FUNCTION_BLOCK Process EXTENDS Station IMPLEMENTS IProcess
VAR_INPUT
END_VAR
VAR_OUTPUT
END_VAR
VAR
	_isProcess : BOOL;
	_startPos : MC_LREAL;
	_endPos : MC_LREAL;
	_processVelo : MC_LREAL;
END_VAR

METHOD PUBLIC  Cycle : BOOL
VAR_INPUT
END_VAR
SUPER^.Cycle();
END_METHOD

PROPERTY EndPosition : MC_LREAL
GET
EndPosition := _endPos;
END_GET
SET
_endPos := EndPosition;
END_SET
END_PROPERTY

PROPERTY IsProcess : BOOL
GET
IsProcess := _isProcess;
END_GET
SET
_isProcess := IsProcess;
END_SET
END_PROPERTY

PROPERTY ProcessVelocity : MC_LREAL
GET
ProcessVelocity := _processVelo;
END_GET
SET
_processVelo := ProcessVelocity;
END_SET
END_PROPERTY

PROPERTY StartPosition : MC_LREAL
GET
StartPosition := _startPos;
END_GET
SET
_startPos := StartPosition;
END_SET
END_PROPERTY

END_FUNCTION_BLOCK

(* stored: Version 1.1.0.1, ProductVersion 3.1.4024.12
   POU Process: Id {5bb3084c-8dc2-4985-92e4-194b505a9bed}, SpecialFunc None
   Method Cycle: Id {848fd251-b5bb-419f-acc7-8914b22a5c9a}
   Property EndPosition: Id {7f4a20d7-f0db-4d2e-987f-1dcaac0ba263}
   Get Get: Id {87faf885-3d96-408c-9e10-b4693bedb554}
   Set Set: Id {03f350b3-edfc-4efc-9080-be45df8aab88}
   Property IsProcess: Id {a052c27a-6963-4165-8ce7-0bc042c34c8d}
   Get Get: Id {f4164ad2-69a7-4e7d-937b-ab9c4f869817}
   Set Set: Id {0dae4abf-34d8-44d5-8e71-ec94152bad0d}
   Property ProcessVelocity: Id {2b95ecf7-a866-474e-93f5-19b6d8e1320a}
   Get Get: Id {25f5b52c-e44e-4bf2-b54e-ddc8a6dd0b98}
   Set Set: Id {6d051eea-51d7-48c9-b4ba-ec2df3b6b6c5}
   Property StartPosition: Id {1d4656dd-6887-469c-a588-d1b0b2352c88}
   Get Get: Id {0aa9c050-e945-4a8f-8702-495f128d5c57}
   Set Set: Id {edfae567-ed6f-497e-adb7-c03f78ecc2d6} *)
